(* IEC 61131-3 sources: cc_kush_rewrite/POUs, 7 files *)

(* ---- GLOBAL.st ---- *)
VAR_GLOBAL
	// Системные ФБ
	PULSE : BLINK;
	PULSE_RTRIG : R_TRIG;

	// Системные флаги
	xStateEmergencyStop : BOOL; // Система была аварийно остановлена
	xStateErrorAcceptIdle : BOOL; // Невозможно принять коэффицент шихтования по заданию оператора - сумма коэффицентов не равна 100
	xStateErrorCheckReady : BOOL; // Проверки стадии готовности к пуску провалились
	xStateAutoWorking : BOOL; // Система полностью запущена и работает в автоматическом режиме
	// Расчёт КИУМ
	ICUR_PRECENT : REAL; // Коэффициент использования установленной мощности (в процентах)
	rElectricityMeter : REAL; // Раход электроэнергии

	// Ограничение производительности
	EFFICIENCY_LIMIT_RATE : REAL := 1; // Коэффицент ограничения производительности (0-1)

	// Переменные симуляции
	SIMULATION : BOOL := TRUE;
	SIMULATION_BUNKER_WEIGHT : BOOL := FALSE; // Включение симуляции расхода и пополнения веса бункеров

	// == MODBUS РЕГИСТРЫ ДЛЯ SCADA ==
	// Массив регистров для передачи данных в SCADA систему
	awModbusInputRegisters : ARRAY [0..511] OF WORD; // Modbus Input регистры
	awModbusHoldingRegisters : ARRAY [0..511] OF WORD; // Modbus Holding регистры

	// == СИГНАЛЫ СВЯЗИ СО SCADA ==
	SCADA_HEARTBEAT : BOOL := FALSE; // Пульсирующий сигнал от SCADA (0 → 1 → 0) для контроля связи

END_VAR
VAR_GLOBAL RETAIN
	// == НАСТРОЙКИ ОСТАНОВКИ ==
	BUNKER_INSTANT_STOP : BOOL := FALSE; // Флаг мгновенной остановки бункеров (TRUE = одновременная остановка всех 3-х бункеров, FALSE = последовательная остановка)

	// == ОПЦИИ ВКЛЮЧЕНИЯ ИСТОЧНИКОВ В ГЛОБАЛЬНУЮ АВАРИЙНУЮ ОСТАНОВКУ ==
	// TRUE = источник включен в цепь глобальной аварийной остановки комплекса
	// FALSE = источник НЕ вызывает глобальную остановку

	// Датчики безопасности
	ENABLE_GLOBAL_ESTOP_ZQ : BOOL := TRUE;       // Датчики схода ленты (ZQ Alarm)
	ENABLE_GLOBAL_ESTOP_HQ : BOOL := TRUE;       // Кабель-тросовые выключатели
	ENABLE_GLOBAL_ESTOP_SQ : BOOL := FALSE;      // Концевики ограждений барабана
	ENABLE_GLOBAL_ESTOP_GS : BOOL := TRUE;      // Заштыбовка
	ENABLE_GLOBAL_ESTOP_YS : BOOL := TRUE;       // Продольный разрыв ленты
	ENABLE_GLOBAL_ESTOP_YE : BOOL := TRUE;       // Металлодетектор
	ENABLE_GLOBAL_ESTOP_QR : BOOL := FALSE;      // Датчики скорости

	// Системные сигналы
	ENABLE_GLOBAL_ESTOP_SCADA_LOSS : BOOL := FALSE;          // Потеря связи со SCADA
	ENABLE_GLOBAL_ESTOP_PROPORTION : BOOL := FALSE;          // Ошибка суммы пропорций
	ENABLE_GLOBAL_ESTOP_MOTOR_CURRENT_HH : BOOL := FALSE;    // Аварийный уровень тока (HH)
	ENABLE_GLOBAL_ESTOP_VFD_FAILURE : BOOL := TRUE;          // Авария VFD (частотного преобразователя)

	// Блокировочные зависимости (глобально)
	ENABLE_GLOBAL_ESTOP_DEPENDENCIES : BOOL := TRUE;         // Блокировочные зависимости между секциями

	// Блокировочные зависимости (индивидуально по секциям)
	// TRUE = секция останавливается при нарушении зависимостей
	// FALSE = секция НЕ останавливается при нарушении зависимостей
	ENABLE_ESTOP_DEPENDENCIES_DUMPER : BOOL := TRUE;         // Зависимости для отвалообразователя
	ENABLE_ESTOP_DEPENDENCIES_CONVEYOR : BOOL := TRUE;       // Зависимости для сборного конвейера
	ENABLE_ESTOP_DEPENDENCIES_BUNKER1 : BOOL := TRUE;        // Зависимости для бункера 1
	ENABLE_ESTOP_DEPENDENCIES_BUNKER2 : BOOL := TRUE;        // Зависимости для бункера 2
	ENABLE_ESTOP_DEPENDENCIES_BUNKER3 : BOOL := TRUE;        // Зависимости для бункера 3

	// == УСТАВКИ ==
	VFD_FREQUENCY_MAX : REAL := 50;
	VFD_FREQUENCY_STEP : REAL := 2;
	VFD_FREQUENCY_INACCURANCY : REAL := 0.5;
	VFD_FREQUENCY_SYNC_TOLERANCE : REAL := 1.5; // Допустимая разница частот для синхронизации моторов

		// == ПАРАМЕТРЫ АЦП/ЦАП ДЛЯ ЧРП ==
	VFD_ADC_MAX : INT := 27648; // Максимальный код АЦП (аналоговый вход/выход)
	VFD_ADC_MIN : INT := 0; // Минимальный код АЦП
	VFD_FREQ_MIN : REAL := 0.0; // Минимальная частота ЧРП (Гц)
	VFD_FREQ_MAX_RANGE : REAL := 50.0; // Максимальная частота для масштабирования АЦП (Гц)

	// == ПАРАМЕТРЫ ТОКА 4-20 мА ==
	VFD_CURRENT_MIN : REAL := 4.0; // Минимальный ток (мА)
	VFD_CURRENT_MAX : REAL := 20.0; // Максимальный ток (мА)
	VFD_CURRENT_ALARM_LL : REAL := 3.8; // Аварийно низкий уровень тока (обрыв линии)
	VFD_CURRENT_ALARM_L : REAL := 4.5; // Низкий уровень тока
	VFD_CURRENT_ALARM_H : REAL := 19.5; // Высокий уровень тока
	VFD_CURRENT_ALARM_HH : REAL := 20.2; // Аварийно высокий уровень тока (перегрузка)

	// == ПАРАМЕТРЫ ДИАПАЗОНА ТЕМПЕРАТУР ==
	TEMP_BEARING_MIN : REAL := 0.0; // Минимальная температура подшипникового узла (°C)
	TEMP_BEARING_MAX : REAL := 100.0; // Максимальная температура подшипникового узла (°C)

	// Настройка виброобрушения
	VIBRATOR_SETTINGS : ST_BunkerVibratorSettings := (
		TIME_ACTIVE := T#15S,
		TIME_PAUSE_VIBRATOR := T#30S,
		TIME_PAUSE_FB := T#30S,
		COUNT_CYCLE := 3
		);

	// Время шага последовательного запуска вибраторов (задержка между запуском каждого следующего вибратора в фазе ACTIVE)
	TIME_VIBRATOR_SEQUENTIAL_START_STEP : TIME := T#4S;

	// Настройка пневмообрушения
	PNEUMO_SETTINGS : ST_BunkerVibratorSettings := (
		TIME_ACTIVE := T#10S,
		TIME_PAUSE_VIBRATOR := T#10S,
		TIME_PAUSE_FB := T#30S,
		COUNT_CYCLE := 3
		);

	// Опция плавного задания частоты
	VFD_SMOOTH_SET_FREQUENCY : BOOL := FALSE;

	// Таймеры последовательного запуска механизмов в автоматическом режиме
	TIME_AFTER_START_DUMPER : TIME := T#120S; // Время ожидания после запуска отвалообразователя
	TIME_AFTER_START_CONVEYOR : TIME := T#120S; // Время ожидания после запуска конвейера
	TIME_AFTER_START_BUNKER_1 : TIME := T#120S; // Время ожидания после запуска бункера 1
	TIME_AFTER_START_BUNKER_2 : TIME := T#120S; // Время ожидания после запуска бункера 2
	TIME_AFTER_START_BUNKER_3 : TIME := T#120S; // Время ожидания после запуска бункера 3

	// Таймеры контроля выполнения команд (тайм-ауты)
	TIME_TIMEOUT_START_DUMPER_CONVEYOR : TIME := T#30S; // Тайм-аут запуска моторов конвейера отвалообразователя (STARTING → WORK)
	TIME_TIMEOUT_START_DUMPER_ROTATION : TIME := T#20S; // Тайм-аут запуска моторов поворота отвалообразователя (STARTING → WORK)
	TIME_TIMEOUT_START_CONVEYOR : TIME := T#30S; // Тайм-аут запуска моторов сборного конвейера (STARTING → WORK)
	TIME_TIMEOUT_START_BUNKER : TIME := T#20S; // Тайм-аут запуска вибропитателей бункера (STARTING → WORK)
	TIME_TIMEOUT_STOP_DUMPER_CONVEYOR : TIME := T#30S; // Тайм-аут остановки моторов конвейера отвалообразователя (STOPPING → IDLE)
	TIME_TIMEOUT_STOP_DUMPER_ROTATION : TIME := T#20S; // Тайм-аут остановки моторов поворота отвалообразователя (STOPPING → IDLE)
	TIME_TIMEOUT_STOP_CONVEYOR : TIME := T#30S; // Тайм-аут остановки моторов сборного конвейера (STOPPING → IDLE)
	TIME_TIMEOUT_STOP_BUNKER : TIME := T#20S; // Тайм-аут остановки вибропитателей бункера (WORK → IDLE)

	// Таймер ожидания восстановления потерянной обратной связи VFD во время работы
	TIME_TIMEOUT_VFD_FEEDBACK_LOST : TIME := T#3S; // Если обратная связь VFD пропала во время WORK и не вернулась в течение этого времени → аварийная остановка

	// Таймер ожидания пропавшего сигнала обратной связи работы механизма
	TIME_WAITING_FEEDBACK : TIME := T#0S;

	// == ПАРАМЕТРЫ СВЯЗИ СО SCADA ==
	SCADA_HEARTBEAT_TIMEOUT : TIME := T#5S; // Таймаут отсутствия изменений heartbeat сигнала (потеря связи)

	// Таймаут контроля суммы пропорций в режиме WORK
	BUNKER_PROPORTION_SUM_TIMEOUT : TIME := T#20S; // Время ожидания корректировки суммы пропорций оператором (сумма должна быть = 100%)

	// Скорость конвейера
	CONVEYOR_DEAFULT_SPEED : REAL := -1;

	// Температура подшипникового узла мотора вибропитателя
	MOTOR_VIBFEEDER_TEMP_POINTS : ST_AlarmSetpoints := (
		LL_Value := -1,
		L_Value := -1,
		H_Value := -1,
		HH_Value := -1);
	// Ток мотора вибропитателя
	MOTOR_VIBFEEDER_CURRENT_POINTS : ST_AlarmSetpoints := (
		LL_Value := -1,
		L_Value := -1,
		H_Value := -1,
		HH_Value := -1);
	// Ток мотора вибратора
	MOTOR_VIBRATOR_CURRENT_POINTS : ST_AlarmSetpoints := (
		LL_Value := -1,
		L_Value := -1,
		H_Value := -1,
		HH_Value := -1);
	// Ток мотора конвейера отвалообразователя
	MOTOR_CONVEYOR_CURRENT_POINTS : ST_AlarmSetpoints := (
		LL_Value := -1,
		L_Value := -1,
		H_Value := -1,
		HH_Value := -1);
	// Ток мотора конвейера сборного
	MOTOR_CONVEYOR_PREFABRICATED_CURRENT_POINTS : ST_AlarmSetpoints := (
		LL_Value := -1,
		L_Value := -1,
		H_Value := -1,
		HH_Value := -1);
	// Ток мотора поворота отвалообразователя
	MOTOR_ROTATION_CURRENT_POINTS : ST_AlarmSetpoints := (
		LL_Value := -1,
		L_Value := -1,
		H_Value := -1,
		HH_Value := -1);

	// Предпусковая сигнализация конвейера отвалообразователя
	DUMPER_CONVEYOR_PRESTART_ALARM_SETTINGS : ST_PreStartAlarmSettings := (
		OPTION_ENABLE := TRUE, // Опция на включение ППЗ в алгоритм
		TIME_FIRST_SIGNAL := T#3S, // Время звучания первого сигнала
		TIME_FIRST_SIGNAL_PAUSE := T#3S, // Пауза после первого сигнала
		TIME_SECOND_SIGNAL := T#3S, // Время звучания второго сигнала
		TIME_SECOND_SIGNAL_PAUSE := T#3S); // Пауза после втотрого сигнала

	// Предпусковая сигнализация сборного конвейера
	CONVEYOR_PRESTART_ALARM_SETTINGS : ST_PreStartAlarmSettings := (
		OPTION_ENABLE := TRUE, // Опция на включение ППЗ в алгоритм
		TIME_FIRST_SIGNAL := T#3S, // Время звучания первого сигнала
		TIME_FIRST_SIGNAL_PAUSE := T#3S, // Пауза после первого сигнала
		TIME_SECOND_SIGNAL := T#3S, // Время звучания второго сигнала
		TIME_SECOND_SIGNAL_PAUSE := T#3S); // Пауза после втотрого сигнала

	// Световая индикация Гц
	ANNUNCIATOR_LIGHT_HZ : REAL := 2;

	// Частота мотора конвейера
	MOTOR_FREQUENCY_CONVEYOR : REAL := 50;
	// Частота мотора конвейера отвалообразователя
	MOTOR_FREQUENCY_DUMPER_CONVEYOR : REAL := 50;
	// Частота мотора поворота отвалообразователя
	MOTOR_FREQUENCY_DUMPER_ROTATION : REAL := -1;

	BUNKER_MINIMAL_WEIGHT :REAL := 0; // Уставка минимального веса бункера. Результат <= считывается алгоритмом как пустой бункер.

	// Уставки бункера
	PNEUMATIC_COLLAPSE_TIME : TIME := T#0S; // Уставка времени таймера пневмообрушения
	BUNKER_WORK_PRECENT_1 : REAL; // Уставка пропорции шихтования для бункера 1
	BUNKER_WORK_PRECENT_2 : REAL; // Уставка пропорции шихтования для бункера 2
	BUNKER_WORK_PRECENT_3 : REAL; // Уставка пропорции шихтования для бункера 3
	BUNKER_VIBFEEDER_START_FREQUENCY : REAL := 10.0; // Минимальная частота для запуска вибропитателей (Гц)
	BUNKER_VIBFEEDER_FREQUENCY_TARGET_SUM : REAL := 50.0; // Целевая суммарная частота вибропитателей (Гц)
    BUNKER_ENABLE_PID : BOOL := FALSE;
    BUNKER_ENABLE_PROPORTION_MONITORING : BOOL := FALSE;

	// == КОНТРОЛЬ МИНИМАЛЬНОЙ И МАКСИМАЛЬНОЙ ЧАСТОТЫ ВИБРОПИТАТЕЛЯ (ДЛЯ ПИД-РЕГУЛЯТОРА) ==
	BUNKER_VIBFEEDER_MIN_FREQUENCY_LIMIT : REAL := 5.0; // Минимальная допустимая частота вибропитателя (Гц) - при достижении этой уставки запускается таймер аварии
	BUNKER_VIBFEEDER_MIN_FREQUENCY_TIMEOUT : TIME := T#30S; // Время задержки перед аварийной остановкой при достижении минимальной частоты
	BUNKER_VIBFEEDER_MAX_FREQUENCY_LIMIT : REAL := 50.0; // Максимальная допустимая частота вибропитателя (Гц) - при достижении этой уставки запускается таймер аварии
	BUNKER_VIBFEEDER_MAX_FREQUENCY_TIMEOUT : TIME := T#30S; // Время задержки перед аварийной остановкой при достижении максимальной частоты

	// Ручное задание частоты на бункер (работает в ручном режиме управления)
	BUNKER_1_FREQ_VIBFEEDER : REAL := 30;
	BUNKER_1_FREQ_VIBRATOR : REAL := 30;
	BUNKER_2_FREQ_VIBFEEDER : REAL := 30;
	BUNKER_2_FREQ_VIBRATOR : REAL := 30;
	BUNKER_3_FREQ_VIBFEEDER : REAL := 30;
	BUNKER_3_FREQ_VIBRATOR : REAL := 30;

	// Светофор бункера
	BUNKER_WEIGHT_LIGHT_RED : REAL := 90; // Уставка веса бункера для красного светофора
	BUNKER_WEIGHT_LIGHT_YELLOW : REAL := 80; // Уставка веса бункера для жёлтого светофора
	BUNKER_WEIGHT_LIGHT_GREEN : REAL := 50; // Уставка веса бункера для зелёного светофора

	BUNKER_WEIGHT_LIGHT_RED_SPECIAL : REAL := 10; // Уставка веса бункера для красного светофора, когда сырье закончилось и требуется остановить подачу материала в остальные бункеры для будущего алгоритма опустошения

	// Константы
	AMOUNT_BUNKER_MOTOR_VIBFEEDER : INT := 2;
	AMOUNT_BUNKER_MOTOR_VIBRATOR : INT := 4;

	// == УСТАВКИ ЗАДЕРЖКИ СРАБАТЫВАНИЯ ДАТЧИКОВ БЕЗОПАСНОСТИ ==
	// Таймеры задержки для датчиков отвалообразователя (Dumper)
	TIME_DELAY_SENSOR_DUMPER_ZQ_ALARM : TIME := T#3S;   // Задержка срабатывания датчика схода ленты (Alarm)
	TIME_DELAY_SENSOR_DUMPER_ZQ_WARNING : TIME := T#0S; // Задержка срабатывания датчика схода ленты (Warning)
	TIME_DELAY_SENSOR_DUMPER_HQ : TIME := T#0S;         // Задержка срабатывания кабель-тросового выключателя
	TIME_DELAY_SENSOR_DUMPER_SQ : TIME := T#0S;         // Задержка срабатывания датчика ограждения барабана
	TIME_DELAY_SENSOR_DUMPER_GS : TIME := T#3S;         // Задержка срабатывания датчика заштыбовки
	TIME_DELAY_SENSOR_DUMPER_YS : TIME := T#3S;         // Задержка срабатывания датчика продольного разрыва
	TIME_DELAY_SENSOR_DUMPER_QR : TIME := T#0S;         // Задержка срабатывания датчика скорости

	// Таймеры задержки для датчиков сборного конвейера (Conveyor)
	TIME_DELAY_SENSOR_CONVEYOR_ZQ_ALARM : TIME := T#3S;   // Задержка срабатывания датчика схода ленты (Alarm)
	TIME_DELAY_SENSOR_CONVEYOR_ZQ_WARNING : TIME := T#0S; // Задержка срабатывания датчика схода ленты (Warning)
	TIME_DELAY_SENSOR_CONVEYOR_HQ : TIME := T#0S;         // Задержка срабатывания кабель-тросового выключателя
	TIME_DELAY_SENSOR_CONVEYOR_SQ : TIME := T#0S;         // Задержка срабатывания датчика ограждения барабана
	TIME_DELAY_SENSOR_CONVEYOR_GS : TIME := T#3S;         // Задержка срабатывания датчика заштыбовки
	TIME_DELAY_SENSOR_CONVEYOR_YS : TIME := T#3S;         // Задержка срабатывания датчика продольного разрыва
	TIME_DELAY_SENSOR_CONVEYOR_YE : TIME := T#0S;         // Задержка срабатывания металлодетектора
	TIME_DELAY_SENSOR_CONVEYOR_QR : TIME := T#0S;         // Задержка срабатывания датчика скорости
END_VAR

(* ---- FB_ConveyorWeight.st ---- *)
FUNCTION_BLOCK FB_ConveyorWeight
VAR_INPUT
	wModbusReg : ARRAY [0..22] OF WORD;
END_VAR
VAR_OUTPUT
	qrWeight : REAL; 			//	0x0 Производительность
	qrSpeed : REAL; 			//	0x2 Скорость
	qrWorkLoad : REAL; 			//	0x4 Погонная нагрузка
	qrVoltageTenso_1 : REAL; 	//	0x6 Текущее напряжение тензодатчика 1
	qrVoltageTenso_2 : REAL; 	//	0x8 Текущее напряжение тензодатчика 2
	qrVoltageTenso_3 : REAL; 	//	0xA Текущее напряжение тензодатчика 3
	qrVoltageTenso_4 : REAL; 	//	0xC Текущее напряжение тензодатчика 4
 	qrCounterShift : REAL;		//	0xE Счётчик: смена
	qrCounterDay : REAL;		//	0xE Счётчик: смена
	qrCounterMonth : REAL;		//	0xE Счётчик: смена
	qrCounterCommon : REAL;		//	0xE Счётчик: смена

END_VAR
VAR
END_VAR

END_FUNCTION_BLOCK

(* ---- FB_DumperControl.st ---- *)
FUNCTION_BLOCK FB_DumperControl
VAR_INPUT
	Dumper : REFERENCE TO ST_Dumper;
	xLocalMode : BOOL; // TRUE = местный режим (ПМУ), FALSE = дистанционный режим (SCADA)
	xStart : BOOL; // Команда запуска отвалообразователя (дистанционный режим)
	xStop : BOOL; // Команда остановки (дистанционный режим)
	xEmergencyStop : BOOL; // Аварийная остановка
	xReset : BOOL; // Сброс в начальное состояние
	xDisableAutoEmergencyStop : BOOL; // Отключение автоматических аварийных остановок по датчикам безопасности
END_VAR
VAR_OUTPUT
	eStage : E_StageWithPreStartAlarm; // Текущая стадия
	eStageToSCADA : E_ScadaStatesDevice; // Передача состояния скаде
END_VAR
VAR
	// Состояния
	STAGE : E_StageWithPreStartAlarm := E_StageWithPreStartAlarm.IDLE;

	// Объединенные команды (ПМУ или SCADA в зависимости от режима)
	xStartCommand : BOOL; // Фактическая команда запуска (из ПМУ или SCADA)
	xStopCommand : BOOL; // Фактическая команда остановки (из ПМУ или SCADA)

	// Целевые частоты для моторов
	rTargetFreqConv1 : REAL := 0.0;
	rTargetFreqConv2 : REAL := 0.0;
	rTargetFreqRot1 : REAL := 0.0;
	rTargetFreqRot2 : REAL := 0.0;

	// Переменные синхронизации моторов конвейера
	xVFDsReady : BOOL; // Оба ЧРП конвейера готовы и запущены
	xFrequenciesSynchronized : BOOL; // Частоты синхронизированы в пределах допуска
	xConditionToProceed : BOOL; // Общее условие для продолжения разгона

	// Подстадии запуска (для последовательного включения тормозов и VFD)
	nStartingSubstage : INT := 0;
	// 0 - RELEASE_BRAKE: Отпускание тормозов
	// 1 - WAIT_BRAKE_FEEDBACK: Ожидание обратной связи тормозов
	// 2 - START_VFD: Запуск VFD
	// 3 - RAMPING: Разгон частоты до рабочей

	// Подстадии остановки (для последовательного выключения VFD и тормозов)
	nStoppingSubstage : INT := 0;
	// 0 - Нормальная работа
	// 1 - SET_FREQUENCY_ZERO: Установка частоты 0 на аналоговый выход
	// 2 - WAIT_FREQUENCY_ZERO: Ожидание подтверждения частоты 0 с аналогового входа
	// 3 - STOP_VFD: Остановка VFD (снятие команды пуска)
	// 4 - WAIT_VFD_STOP: Ожидание остановки VFD (обратная связь)
	// 5 - ACTIVATE_BRAKE: Активация тормозов
	// 6 - WAIT_BRAKE_FEEDBACK: Ожидание обратной связи тормозов

	// Состояние схемы контакторов (TRUE = схема собрана, FALSE = схема разобрана)
	xCircuitBuilt : BOOL := FALSE;
	xCircuitBuiltRotation : BOOL := FALSE;

	// Таймеры контроля выполнения команд
	fbTimerStarting : TON; // Тайм-аут запуска (STARTING → WORK)
	fbTimerStopping : TON; // Тайм-аут остановки (WORK → IDLE)
	fbTimerRotation : TON; // Тайм-аут выполнения команд поворота
	// Таймер на работу тормоза
	tonTimerEnableBreakerConveyor : TON; // Задержка включения тормоза на конвейере
	tonTimerEnableBreakerRotation : TON; // Задержка включения тормоза на повороте

	// == Управление поворотом ==
	xRotationLeftActive : BOOL; // Поворот влево активен
	xRotationRightActive : BOOL; // Поворот вправо активен
	nRotationSubstage : INT := 0; // Подстадии поворота
	// 0 - IDLE: Нет активного поворота
	// 1 - RELEASE_BRAKE: Отпускание тормоза поворота
	// 2 - WAIT_BRAKE_FEEDBACK: Ожидание обратной связи тормоза
	// 3 - START_VFD: Запуск VFD поворота
	// 4 - WORKING: Моторы поворота работают
	// 5 - SET_FREQUENCY_ZERO: Установка частоты 0 на аналоговый выход
	// 6 - WAIT_FREQUENCY_ZERO: Ожидание подтверждения частоты 0 с аналогового входа
	// 7 - STOP_VFD: Остановка VFD поворота (снятие команды пуска)
	// 8 - WAIT_VFD_STOP: Ожидание остановки VFD (обратная связь)
	// 9 - ACTIVATE_BRAKE: Активация тормоза

	simInit : BOOL;
	i : INT;
END_VAR

// ========================================
// FB_DumperControl - Управление отвалообразователем
// ========================================
//
// РЕЖИМЫ УПРАВЛЕНИЯ:
//
// 1. МЕСТНЫЙ РЕЖИМ (xLocalMode = TRUE):
//    - Команды берутся с кнопок ПМУ (Dumper.fbBtnStart, fbBtnStop)
//    - Конвейер: ПУСК/СТОП по фронтам кнопок
//    - Поворот: работает пока кнопка ЗАЖАТА (fbBtnTurnLeft/Right)
//    - Автоматически устанавливает eStateRemote = Manual
//
// 2. ДИСТАНЦИОННЫЙ РЕЖИМ (xLocalMode = FALSE):
//    - Команды берутся из входов ФБ (xStart, xStop)
//    - Конвейер: ПУСК/СТОП по входам ФБ
//    - Поворот: импульсные команды через Dumper.cmdTurnLeft/Right/Stop
//    - Режим устанавливается через SCADA (Manual/Remote/Auto)
//
// УПРАВЛЕНИЕ КОНВЕЙЕРОМ:
// - ПУСК: включение конвейеров отвалообразователя
// - СТОП: плавная остановка с последовательным выключением VFD и тормозов
//
// УПРАВЛЕНИЕ ПОВОРОТОМ:
// - Местный: поворот пока кнопка зажата (отпустили - остановка)
// - Дистанционный: импульсные команды от SCADA
// - Блокировка по концевикам (fbEndSwitchLeft/Right):
//   * Если концевик сработал (qxSignal = FALSE), команда поворота в эту сторону игнорируется
//   * Поворот автоматически останавливается при достижении концевика
//
// ========================================

// ========================================
// ИНИЦИАЛИЗАЦИЯ СИГНАЛОВ
// ========================================

// ПМУ - СТАРТ
Dumper.fbBtnStart(
	ixSignal := , // Подключить физический вход
	xEnableRattlingFilter := TRUE,
	tStabilityTime := T#100MS
);

// ПМУ - СТОП
Dumper.fbBtnStop(
	ixSignal := , // Подключить физический вход
	xEnableRattlingFilter := TRUE,
	tStabilityTime := T#100MS
);

// ПМУ - Аварийная остановка
Dumper.fbBtnEmergencyStop(
	ixSignal := , // Подключить физический вход
	xEnableRattlingFilter := TRUE,
	tStabilityTime := T#100MS
);

// ПМУ Поворот влево/вправо
Dumper.fbBtnTurnLeft(
	ixSignal := , // Подключить физический вход
	xEnableRattlingFilter := TRUE,
	tStabilityTime := T#100MS
);

Dumper.fbBtnTurnRight(
	ixSignal := , // Подключить физический вход
	xEnableRattlingFilter := TRUE,
	tStabilityTime := T#100MS
);

Dumper.fbEndSwitchLeft(
	ixSignal := , // Подключить физический вход
	xEnableRattlingFilter := TRUE,
	tStabilityTime := T#100MS
);

Dumper.fbEndSwitchRight(
	ixSignal := , // Подключить физический вход
	xEnableRattlingFilter := TRUE,
	tStabilityTime := T#100MS
);

// Сигналы тормозоов (Обратная связь)
Dumper.fbBreakerConveyor(
	ixSignal := , // Физ. сигнал
	xEnableRattlingFilter := TRUE);

Dumper.fbBreakerRotation(
	ixSignal := , // Физ. сигнал
	xEnableRattlingFilter := TRUE);

// Двигатели конвейера
FOR i := 1 TO 2 BY 1 DO
	Dumper.MotorConveyor[i].fbStateKM(
		ixSignal := , // Состояние контактора
		xEnableRattlingFilter := TRUE
	);

	Dumper.MotorConveyor[i].fbStatorOverheat(
		ixSignal := , // Перегрев статора
		xEnableRattlingFilter := TRUE
	);

	Dumper.MotorConveyor[i].fbStateQF(
		ixSignal := , // Автомат. выключатель
		xEnableRattlingFilter := TRUE
	);

	Dumper.MotorConveyor[i].VFD.fbStateFailure(
		ixSignal := , // ЧРП - ошибка
		xEnableRattlingFilter := TRUE
	);

	Dumper.MotorConveyor[i].VFD.fbStateRdyToStart(
		ixSignal := , // ЧРП - Готовность
		xEnableRattlingFilter := TRUE
	);

	Dumper.MotorConveyor[i].VFD.fbStateIsWorking(
		ixSignal := , // ЧРП - Работа
		xEnableRattlingFilter := TRUE
	);

	// Инициализация устройств
	Dumper.MotorConveyor[i].Device(
		ixFeedback := Dumper.MotorConveyor[i].fbStateKM.qxSignal,
		xEnableFeedback := TRUE
	);

	// ЧРП
	Dumper.MotorConveyor[i].VFD.Device(
		ixFeedback := Dumper.MotorConveyor[i].VFD.fbStateIsWorking.qxSignal,
		xEnableFeedback := TRUE
	);

	// VFD.qxStart теперь управляется напрямую в алгоритме (TRUE = ПУСК, FALSE = СТОП)

	// Диагностика тока
	Dumper.MotorConveyor[i].VFD.fbRangeDiagnostic(
		irValue := Dumper.MotorConveyor[i].VFD.wMotorCurrent.rTag,
		irSetpointL := MOTOR_CONVEYOR_CURRENT_POINTS.L_Value,
		irSetpointLL := MOTOR_CONVEYOR_CURRENT_POINTS.LL_Value,
		irSetpointH := MOTOR_CONVEYOR_CURRENT_POINTS.H_Value,
		irSetpointHH := MOTOR_CONVEYOR_CURRENT_POINTS.HH_Value,
		ixEnable := TRUE
	);

	// Аналоговый вход ЧРП (чтение текущей частоты)
	Dumper.MotorConveyor[i].VFD.fbAnalogInput(
		xSimulation := SIMULATION,
		iADC_Code := Dumper.MotorConveyor[i].VFD.nActualFrequencyADC,
		refEngValue := Dumper.MotorConveyor[i].VFD.rActualFrequency,
		refSimValue := Dumper.MotorConveyor[i].VFD.rSimulatedFrequency,
		rAlarm_LL := VFD_CURRENT_ALARM_LL,
		rAlarm_L := VFD_CURRENT_ALARM_L,
		rAlarm_H := VFD_CURRENT_ALARM_H,
		rAlarm_HH := VFD_CURRENT_ALARM_HH,
		iADC_Max := VFD_ADC_MAX,
		iADC_Min := VFD_ADC_MIN,
		rEngValue_Max := VFD_FREQ_MAX_RANGE,
		rEngValue_Min := VFD_FREQ_MIN,
		rCurrent_Max := VFD_CURRENT_MAX,
		rCurrent_Min := VFD_CURRENT_MIN
	);

	// Аналоговый выход ЧРП (задание частоты)
	Dumper.MotorConveyor[i].VFD.fbAnalogOutput(
		xEnable := Dumper.MotorConveyor[i].VFD.Device.qxActive,
		rEngValue := Dumper.MotorConveyor[i].VFD.Frequency.qrCurrentFrequency,
		rEngValue_Max := VFD_FREQ_MAX_RANGE,
		rEngValue_Min := VFD_FREQ_MIN,
		rCurrent_Max := VFD_CURRENT_MAX,
		rCurrent_Min := VFD_CURRENT_MIN,
		iDAC_Max := VFD_ADC_MAX,
		iDAC_Min := VFD_ADC_MIN,
		rAlarm_LL := VFD_CURRENT_ALARM_LL,
		rAlarm_L := VFD_CURRENT_ALARM_L,
		rAlarm_H := VFD_CURRENT_ALARM_H,
		rAlarm_HH := VFD_CURRENT_ALARM_HH,
		xEnableClamp := TRUE
	);
	Dumper.MotorConveyor[i].VFD.nSetOutSignalToModule := Dumper.MotorConveyor[i].VFD.fbAnalogOutput.iDAC_Code;
END_FOR;

// Двигатели поворота
FOR i := 1 TO 2 BY 1 DO
	Dumper.MotorRotation[i].fbStateKM(
		ixSignal := , // Состояние контактора
		xEnableRattlingFilter := TRUE
	);

	Dumper.MotorRotation[i].fbStatorOverheat(
		ixSignal := , // Перегрев статора
		xEnableRattlingFilter := TRUE
	);

	Dumper.MotorRotation[i].fbStateQF(
		ixSignal := , // Автомат. выключатель
		xEnableRattlingFilter := TRUE
	);

	Dumper.MotorRotation[i].VFD.fbStateFailure(
		ixSignal := , // ЧРП - ошибка
		xEnableRattlingFilter := TRUE
	);

	Dumper.MotorRotation[i].VFD.fbStateRdyToStart(
		ixSignal := , // ЧРП - Готовность
		xEnableRattlingFilter := TRUE
	);

	Dumper.MotorRotation[i].VFD.fbStateIsWorking(
		ixSignal := , // ЧРП - Работа
		xEnableRattlingFilter := TRUE
	);

	Dumper.MotorRotation[i].fbRotationStatus(
		ixSignal := , // Статус вращения
		xEnableRattlingFilter := TRUE
	);

	// Инициализация устройств
	Dumper.MotorRotation[i].Device(
		ixFeedback := Dumper.MotorRotation[i].fbStateKM.qxSignal,
		xEnableFeedback := TRUE
	);

	// ЧРП
	Dumper.MotorRotation[i].VFD.Device(
		ixFeedback := Dumper.MotorRotation[i].VFD.fbStateIsWorking.qxSignal,
		xEnableFeedback := TRUE
	);

	// VFD.qxStart теперь управляется напрямую в алгоритме (TRUE = ПУСК, FALSE = СТОП)

	// Диагностика тока
	Dumper.MotorRotation[i].VFD.fbRangeDiagnostic(
		irValue := Dumper.MotorRotation[i].VFD.wMotorCurrent.rTag,
		irSetpointL := MOTOR_ROTATION_CURRENT_POINTS.L_Value,
		irSetpointLL := MOTOR_ROTATION_CURRENT_POINTS.LL_Value,
		irSetpointH := MOTOR_ROTATION_CURRENT_POINTS.H_Value,
		irSetpointHH := MOTOR_ROTATION_CURRENT_POINTS.HH_Value,
		ixEnable := TRUE
	);

	// Аналоговый вход ЧРП (чтение текущей частоты)
	Dumper.MotorRotation[i].VFD.fbAnalogInput(
		xSimulation := SIMULATION,
		iADC_Code := Dumper.MotorRotation[i].VFD.nActualFrequencyADC,
		refEngValue := Dumper.MotorRotation[i].VFD.rActualFrequency,
		refSimValue := Dumper.MotorRotation[i].VFD.rSimulatedFrequency,
		rAlarm_LL := VFD_CURRENT_ALARM_LL,
		rAlarm_L := VFD_CURRENT_ALARM_L,
		rAlarm_H := VFD_CURRENT_ALARM_H,
		rAlarm_HH := VFD_CURRENT_ALARM_HH,
		iADC_Max := VFD_ADC_MAX,
		iADC_Min := VFD_ADC_MIN,
		rEngValue_Max := VFD_FREQ_MAX_RANGE,
		rEngValue_Min := VFD_FREQ_MIN,
		rCurrent_Max := VFD_CURRENT_MAX,
		rCurrent_Min := VFD_CURRENT_MIN
	);

	// Аналоговый выход ЧРП (задание частоты)
	Dumper.MotorRotation[i].VFD.fbAnalogOutput(
		xEnable := Dumper.MotorRotation[i].VFD.Device.qxActive,
		rEngValue := Dumper.MotorRotation[i].VFD.Frequency.qrCurrentFrequency,
		rEngValue_Max := VFD_FREQ_MAX_RANGE,
		rEngValue_Min := VFD_FREQ_MIN,
		rCurrent_Max := VFD_CURRENT_MAX,
		rCurrent_Min := VFD_CURRENT_MIN,
		iDAC_Max := VFD_ADC_MAX,
		iDAC_Min := VFD_ADC_MIN,
		rAlarm_LL := VFD_CURRENT_ALARM_LL,
		rAlarm_L := VFD_CURRENT_ALARM_L,
		rAlarm_H := VFD_CURRENT_ALARM_H,
		rAlarm_HH := VFD_CURRENT_ALARM_HH,
		xEnableClamp := TRUE
	);
	Dumper.MotorRotation[i].VFD.nSetOutSignalToModule := Dumper.MotorRotation[i].VFD.fbAnalogOutput.iDAC_Code;
END_FOR;

// Датчики безопасности
FOR i := 1 TO 4 BY 1 DO
	Dumper.fbZQAlarm[i](
		ixSignal := ,
		xEnableRattlingFilter := TRUE
	);

	Dumper.fbZQWarning[i](
		ixSignal := ,
		xEnableRattlingFilter := TRUE
	);

	Dumper.fbHQ_IsOk[i](
		ixSignal := ,
		xEnableRattlingFilter := TRUE
	);
END_FOR;

FOR i := 1 TO 2 BY 1 DO
	Dumper.fbSQ_IsOk[i](
		ixSignal := ,
		xEnableRattlingFilter := TRUE
	);

	Dumper.fbQR[i](
		ixSignal := ,
		xEnableRattlingFilter := FALSE // Только edge detection
	);
END_FOR;

Dumper.fbGS1(
	ixSignal := ,
	xEnableRattlingFilter := TRUE
);

Dumper.fbYS1(
	ixSignal := ,
	xEnableRattlingFilter := TRUE
);

// ========================================
// ПРЕДПУСКОВАЯ СИГНАЛИЗАЦИЯ
// ========================================

Dumper.fbPreStartAlarm(
	ixStart := STAGE = PRESTART_ALARM,
	ixStop := xStopCommand OR xReset,
	itFirstSignal := DUMPER_CONVEYOR_PRESTART_ALARM_SETTINGS.TIME_FIRST_SIGNAL,
	itPauseAfterFirst := DUMPER_CONVEYOR_PRESTART_ALARM_SETTINGS.TIME_FIRST_SIGNAL_PAUSE,
	itSecondSignal := DUMPER_CONVEYOR_PRESTART_ALARM_SETTINGS.TIME_SECOND_SIGNAL,
	itPauseAfterSecond := DUMPER_CONVEYOR_PRESTART_ALARM_SETTINGS.TIME_SECOND_SIGNAL_PAUSE,
	qxAlarmPower => Dumper.xHLA
);

// Световая сигнализация во время активной работы поворота
// xHLA включается как при предпусковой сигнализации, так и при повороте
Dumper.xHLA := Dumper.fbPreStartAlarm.qxAlarmPower OR (nRotationSubstage = 4);

Dumper.xStateEnable := STAGE = E_StageWithPreStartAlarm.WORK;
Dumper.xStateStarting := STAGE = E_StageWithPreStartAlarm.STARTING OR STAGE = PRESTART_ALARM;

// ========================================
// ОПРЕДЕЛЕНИЕ СОСТОЯНИЙ ДЛЯ SCADA
// ========================================

// Проверка ошибок оборудования
IF FC_Dumper_GetErrorCommon(Dumper := Dumper) THEN
	Dumper.xStateFailure := TRUE;
END_IF;

// Проверка предупреждений:
// 1. Датчики схода ленты ZQ - уровень Warning
// 2. Контроль тока моторов - уровень L или H
Dumper.xStateWarning := NOT Dumper.fbZQWarning[1].qxSignal
                     OR NOT Dumper.fbZQWarning[2].qxSignal
                     OR NOT Dumper.fbZQWarning[3].qxSignal
                     OR NOT Dumper.fbZQWarning[4].qxSignal
                     OR Dumper.MotorConveyor[1].VFD.fbRangeDiagnostic.qxWarningActive
                     OR Dumper.MotorConveyor[2].VFD.fbRangeDiagnostic.qxWarningActive
                     OR Dumper.MotorRotation[1].VFD.fbRangeDiagnostic.qxWarningActive
                     OR Dumper.MotorRotation[2].VFD.fbRangeDiagnostic.qxWarningActive;

// ========================================
// ОБРАБОТКА ОСТАНОВКИ И СБРОСА
// ========================================

// Сброс в начальное состояние
IF xReset THEN
	Dumper.xStateFailure := FALSE;
END_IF

// Штатная остановка - запускается при получении команды xStop
// Обрабатывается через подстадии в режиме WORK

// ========================================
// ВЫБОР ИСТОЧНИКА КОМАНД (ПМУ ИЛИ SCADA)
// ========================================

// В местном режиме (xLocalMode = TRUE) - команды берутся с ПМУ (кнопки)
// В дистанционном режиме (xLocalMode = FALSE) - команды берутся из SCADA (входы ФБ)
IF xLocalMode THEN
	// Местный режим - команды с ПМУ
	xStartCommand := Dumper.fbBtnStart.qxRisingEdge; // ПУСК по фронту кнопки
	xStopCommand := Dumper.fbBtnStop.qxRisingEdge;   // СТОП по фронту кнопки
ELSE
	// Дистанционный режим - команды из SCADA
	xStartCommand := xStart;
	xStopCommand := xStop;
END_IF;

// ========================================
// АВТОМАТ ПУСКА ОТВАЛООБРАЗОВАТЕЛЯ
// ========================================

// ПРИОРИТЕТНАЯ ПРОВЕРКА АВАРИЙНОЙ ОСТАНОВКИ
// Аварийная остановка имеет наивысший приоритет и срабатывает в любой стадии
// 1. Внешний сигнал аварийной остановки (от SCADA или системы)
// 2. Кнопка аварийной остановки на ПМУ (NC контакт: FALSE = кнопка нажата)
IF xEmergencyStop OR NOT Dumper.fbBtnEmergencyStop.qxSignal THEN
	STAGE := E_StageWithPreStartAlarm.ERROR;
END_IF;

// КРИТИЧЕСКИЕ ОШИБКИ ДАТЧИКОВ БЕЗОПАСНОСТИ
// При срабатывании датчиков безопасности немедленная аварийная остановка,
// если секция НЕ в IDLE (т.е. находится в процессе работы или запуска)
// Блокируется через вход xDisableAutoEmergencyStop
IF FC_Dumper_GetErrorSensors(Dumper := Dumper)
   AND STAGE <> E_StageWithPreStartAlarm.IDLE
   AND NOT xDisableAutoEmergencyStop
THEN
	STAGE := E_StageWithPreStartAlarm.ERROR;
END_IF;

// ПРОВЕРКА ТАЙМ-АУТОВ ВЫПОЛНЕНИЯ КОМАНД
// Тайм-аут запуска: не удалось запустить секцию за установленное время
IF fbTimerStarting.Q THEN
	STAGE := E_StageWithPreStartAlarm.ERROR;
END_IF;

// Тайм-аут остановки: не удалось остановить секцию за установленное время
IF fbTimerStopping.Q THEN
	STAGE := E_StageWithPreStartAlarm.ERROR;
END_IF;

// Тайм-аут поворота: не удалось выполнить команду поворота за установленное время
IF fbTimerRotation.Q THEN
	STAGE := E_StageWithPreStartAlarm.ERROR;
	nRotationSubstage := 0; // Сброс подстадии поворота
END_IF;

CASE STAGE OF
	E_StageWithPreStartAlarm.IDLE:
		// Сброс целевой частоты
		rTargetFreqConv1 := 0.0;
		rTargetFreqConv2 := 0.0;
		rTargetFreqRot1 := 0.0;
		rTargetFreqRot2 := 0.0;

		// Сброс подстадий запуска и остановки
		nStartingSubstage := 0;
		nStoppingSubstage := 0;

		// Сброс таймеров запуска и остановки
		fbTimerStarting(IN := FALSE);
		fbTimerStopping(IN := FALSE);

		// Тормоза активны (удерживают механизм)
		Dumper.qxBreakerConveyor := FALSE;

		IF xStartCommand THEN
			STAGE := PRESTART_ALARM;
		END_IF;

	PRESTART_ALARM:
		// Проверка команды остановки во время предпусковой сигнализации
		IF xStopCommand THEN
			// Прервать предпусковую сигнализацию и вернуться в IDLE
			STAGE := E_StageWithPreStartAlarm.IDLE;
		ELSIF Dumper.fbPreStartAlarm.qxComplete THEN
			STAGE := E_StageWithPreStartAlarm.STARTING;
		END_IF;

	E_StageWithPreStartAlarm.STARTING:
		// Проверка команды остановки во время запуска
		IF xStopCommand THEN
			// Прервать запуск и перейти к процедуре остановки
			STAGE := E_StageWithPreStartAlarm.WORK;
			nStartingSubstage := 0;
			nStoppingSubstage := 1; // Начать процедуру остановки
			fbTimerStarting(IN := FALSE); // Сброс таймера
		END_IF;

		// Таймер ожидания полного запуска секции
		fbTimerStarting(
			IN := TRUE,
			PT := TIME_AFTER_START_DUMPER
		);

		// Последовательный запуск: Тормоза → Обратная связь → VFD → Разгон
		CASE nStartingSubstage OF
			0: // RELEASE_BRAKE - Отпускание тормозов
				// Включить сигнал тормоза (1 = тормоз отпущен)
				Dumper.qxBreakerConveyor := TRUE;
				Dumper.qxBreakerRotation := TRUE;

				// Переход к следующей подстадии
				nStartingSubstage := 1;

			1: // WAIT_BRAKE_FEEDBACK - Ожидание обратной связи тормозов
				// Получить обратную связь реле тормоза
				IF Dumper.fbBreakerConveyor.qxSignal THEN
					// Обратная связь получена, переходим к запуску VFD
					nStartingSubstage := 2;
				END_IF;

			2: // START_VFD - Запуск VFD (контакторы управляются отдельно через cmdBuildCircuitOn/Off)
				// Команда ПУСК на частотный преобразователь (TRUE = ПУСК)
				Dumper.MotorConveyor[1].VFD.qxStart := TRUE;
				Dumper.MotorConveyor[2].VFD.qxStart := TRUE;

				// Установка целевой частоты
				// (FB_FrequencyControl автоматически выберет плавный или прямой пуск через irStep)
				rTargetFreqConv1 := MOTOR_FREQUENCY_DUMPER_CONVEYOR;
				rTargetFreqConv2 := MOTOR_FREQUENCY_DUMPER_CONVEYOR;

				// Если оба VFD запущены (обратная связь), переходим к следующей подстадии
				IF Dumper.MotorConveyor[1].VFD.fbStateIsWorking.qxSignal
					AND Dumper.MotorConveyor[2].VFD.fbStateIsWorking.qxSignal
				THEN
					IF VFD_SMOOTH_SET_FREQUENCY THEN
						// Плавный пуск: переходим к разгону
						nStartingSubstage := 3;
					ELSE
						// Прямой пуск: сразу в режим WORK (частота уже установлена через большой шаг)
						STAGE := E_StageWithPreStartAlarm.WORK;
						nStartingSubstage := 0;
						fbTimerStarting(IN := FALSE); // Сброс таймера
					END_IF;
				END_IF;

			3: // RAMPING - Разгон частоты до рабочей
				// Команды запуска VFD остаются активными (TRUE = ПУСК)
				Dumper.MotorConveyor[1].VFD.qxStart := TRUE;
				Dumper.MotorConveyor[2].VFD.qxStart := TRUE;

				// Задание целевой частоты (передается в FB_FrequencyControl)
				rTargetFreqConv1 := MOTOR_FREQUENCY_DUMPER_CONVEYOR;
				rTargetFreqConv2 := MOTOR_FREQUENCY_DUMPER_CONVEYOR;

				// Переход в режим WORK при достижении целевой частоты
				// Используется регулирование частоты с синхронизацией
				IF Dumper.MotorConveyor[1].VFD.rActualFrequency >= MOTOR_FREQUENCY_DUMPER_CONVEYOR - VFD_FREQUENCY_INACCURANCY
					AND Dumper.MotorConveyor[2].VFD.rActualFrequency >= MOTOR_FREQUENCY_DUMPER_CONVEYOR - VFD_FREQUENCY_INACCURANCY
				THEN
					STAGE := E_StageWithPreStartAlarm.WORK;
					nStartingSubstage := 0; // Сброс для следующего запуска
					fbTimerStarting(IN := FALSE); // Сброс таймера
				END_IF;
		END_CASE;

	E_StageWithPreStartAlarm.WORK:
		// Нормальная работа или штатная остановка через подстадии
		CASE nStoppingSubstage OF
			0: // Нормальная работа
				// Сброс таймера остановки
				fbTimerStopping(IN := FALSE);

				// Обновление целевой частоты конвейера в ручном режиме
				IF Dumper.eStateRemote = E_StateRemote.Manual THEN
					rTargetFreqConv1 := MOTOR_FREQUENCY_DUMPER_CONVEYOR;
					rTargetFreqConv2 := MOTOR_FREQUENCY_DUMPER_CONVEYOR;
				END_IF;

				IF xStopCommand THEN
					// Начать штатную остановку
					nStoppingSubstage := 1;
				END_IF;

			1: // SET_FREQUENCY_ZERO - Установка частоты 0 на аналоговый выход
				// Запуск таймера остановки (тайм-аут на остановку секции)
				fbTimerStopping(
					IN := TRUE,
					PT := TIME_TIMEOUT_STOP_DUMPER
				);

				// Установить целевую частоту 0
				// (FB_FrequencyControl автоматически выберет плавную или прямую остановку через irStep)
				rTargetFreqConv1 := 0.0;
				rTargetFreqConv2 := 0.0;
				rTargetFreqRot1 := 0.0;
				rTargetFreqRot2 := 0.0;

				// Команды пуска VFD остаются активными (TRUE = ПУСК)
				// VFD продолжают работать, но частота снижается
				Dumper.MotorConveyor[1].VFD.qxStart := FALSE; // TODO ВРЕМЕННО
				Dumper.MotorConveyor[2].VFD.qxStart := FALSE;

				// Переход к следующей подстадии
				nStoppingSubstage := 2;

			2: // WAIT_FREQUENCY_ZERO - Ожидание подтверждения частоты 0 с аналогового входа
				// Ждём, пока фактическая частота (с аналогового входа) не снизится до 0 (+/- 2 Гц)
				IF Dumper.MotorConveyor[1].VFD.rActualFrequency <= 2.0
					AND Dumper.MotorConveyor[2].VFD.rActualFrequency <= 2.0
				THEN
					// Частота подтверждена на 0, переходим к остановке VFD
					nStoppingSubstage := 3;
				END_IF;

			3: // STOP_VFD - Остановка VFD (снятие команды пуска)
				// Отключить команду пуска на VFD (FALSE = СТОП)
				Dumper.MotorConveyor[1].VFD.qxStart := FALSE;
				Dumper.MotorConveyor[2].VFD.qxStart := FALSE;

				// Переход к ожиданию обратной связи VFD
				nStoppingSubstage := 4;

			4: // WAIT_VFD_STOP - Ожидание остановки VFD (обратная связь)
				// Проверить обратную связь VFD о выключении
				IF NOT Dumper.MotorConveyor[1].VFD.fbStateIsWorking.qxSignal
					AND NOT Dumper.MotorConveyor[2].VFD.fbStateIsWorking.qxSignal
				THEN
					// VFD выключены, переход к активации тормозов
					nStoppingSubstage := 5;
				END_IF;

			5: // ACTIVATE_BRAKE - Активация тормозов
				// Включение таймера на задержку тормоза
				tonTimerEnableBreakerConveyor(IN:= TRUE, PT:=T#5S);

				IF tonTimerEnableBreakerConveyor.Q THEN // Снять сигнал с тормоза после таймера (поставить на тормоз: FALSE = активен)
					Dumper.qxBreakerConveyor := FALSE;
					Dumper.qxBreakerRotation := FALSE;
					tonTimerEnableBreakerConveyor(IN:= FALSE);
					// Переход к завершению остановки
					nStoppingSubstage := 6;
				END_IF;
			6: // WAIT_BRAKE_FEEDBACK - Переход в IDLE
				// Сброс таймера остановки (успешная остановка)
				fbTimerStopping(IN := FALSE);

				STAGE := E_StageWithPreStartAlarm.IDLE;
				nStoppingSubstage := 0;
		END_CASE;

	E_StageWithPreStartAlarm.ERROR:
		// Состояние ошибки - аварийная остановка и ожидание сброса
		// (используется при серьезных неисправностях, не для штатной остановки)

		// Аварийная остановка: команда СТОП на VFD (FALSE = СТОП)
		Dumper.MotorConveyor[1].VFD.qxStart := FALSE;
		Dumper.MotorConveyor[2].VFD.qxStart := FALSE;
		Dumper.MotorRotation[1].VFD.qxStart := FALSE;
		Dumper.MotorRotation[2].VFD.qxStart := FALSE;
		Dumper.MotorRotation[1].qxVFDReverseStart := FALSE;
		Dumper.MotorRotation[2].qxVFDReverseStart := FALSE;

		// Сброс целевых частот
		rTargetFreqConv1 := 0.0;
		rTargetFreqConv2 := 0.0;
		rTargetFreqRot1 := 0.0;
		rTargetFreqRot2 := 0.0;

		// Активировать тормоза
		Dumper.qxBreakerConveyor := FALSE;
		Dumper.qxBreakerRotation := FALSE;

		// Разборка схем контакторов (аварийная остановка)
		IF Dumper.eStateRemote = E_StateRemote.Auto THEN
			xCircuitBuilt := FALSE;
			xCircuitBuiltRotation := FALSE;
		END_IF;
		// Сброс подстадий для следующего запуска
		nStartingSubstage := 0;
		nStoppingSubstage := 0;
		nRotationSubstage := 0;

		// Сброс таймеров
		fbTimerStarting(IN := FALSE);
		fbTimerStopping(IN := FALSE);
		fbTimerRotation(IN := FALSE);
		tonTimerEnableBreakerConveyor(IN := FALSE);
		tonTimerEnableBreakerRotation(IN:= FALSE);
		// Контакторы управляются отдельно через импульсные команды
		// cmdBuildCircuitOn/Off (см. секцию УПРАВЛЕНИЕ КОНТАКТОРАМИ)

		// Сброс ошибки и переход в IDLE при отсутствии ошибок
		// Для выхода из ERROR требуется:
		// 1. Команда сброса (xReset)
		// 2. Снятие сигнала аварийной остановки (NOT xEmergencyStop)
		// 3. Кнопка аварийной остановки отпущена (NC контакт: TRUE = кнопка отпущена)
		// 4. Отсутствие ошибок оборудования (NOT Dumper.xStateFailure)
		IF xReset AND NOT xEmergencyStop AND Dumper.fbBtnEmergencyStop.qxSignal AND NOT Dumper.xStateFailure THEN
			STAGE := E_StageWithPreStartAlarm.IDLE;
		END_IF
END_CASE;

// ========================================
// ПРОВЕРКА СИНХРОНИЗАЦИИ МОТОРОВ КОНВЕЙЕРА
// ========================================

// Проверка что оба ЧРП конвейера готовы и запущены (обратная связь)
xVFDsReady := Dumper.MotorConveyor[1].VFD.fbStateIsWorking.qxSignal
           AND Dumper.MotorConveyor[2].VFD.fbStateIsWorking.qxSignal;

// Проверка синхронизации текущих частот (разница не превышает допуск)
xFrequenciesSynchronized := ABS(Dumper.MotorConveyor[1].VFD.Frequency.qrCurrentFrequency
                              - Dumper.MotorConveyor[2].VFD.Frequency.qrCurrentFrequency)
                              <= VFD_FREQUENCY_SYNC_TOLERANCE;

// Общее условие для продолжения плавного разгона
// Разгон продолжается только если оба ЧРП запущены И частоты синхронизированы
xConditionToProceed := xVFDsReady AND xFrequenciesSynchronized;

// ========================================
// ОБРАБОТКА ЧАСТОТЫ (после установки целевых значений в CASE)
// ========================================

// Моторы конвейера
Dumper.MotorConveyor[1].VFD.Frequency(
	irMaxFrequency := VFD_FREQUENCY_MAX,
	// Если плавный пуск - используем шаг, иначе - большой шаг для мгновенной установки
	irStep := SEL(VFD_SMOOTH_SET_FREQUENCY, VFD_FREQ_MAX_RANGE, VFD_FREQUENCY_STEP),
	rTargetFrequency := rTargetFreqConv1,
	xPulse := PULSE_RTRIG.Q,
	xConditionToProceed := xConditionToProceed // Синхронизация с мотором 2
);
// qrCurrentFrequency передается напрямую в fbAnalogOutput.rEngValue

Dumper.MotorConveyor[2].VFD.Frequency(
	irMaxFrequency := VFD_FREQUENCY_MAX,
	// Если плавный пуск - используем шаг, иначе - большой шаг для мгновенной установки
	irStep := SEL(VFD_SMOOTH_SET_FREQUENCY, VFD_FREQ_MAX_RANGE, VFD_FREQUENCY_STEP),
	rTargetFrequency := rTargetFreqConv2,
	xPulse := PULSE_RTRIG.Q,
	xConditionToProceed := xConditionToProceed // Синхронизация с мотором 1
);
// qrCurrentFrequency передается напрямую в fbAnalogOutput.rEngValue

// Моторы поворота
Dumper.MotorRotation[1].VFD.Frequency(
	irMaxFrequency := VFD_FREQUENCY_MAX,
	// Если плавный пуск - используем шаг, иначе - большой шаг для мгновенной установки
	irStep := SEL(VFD_SMOOTH_SET_FREQUENCY, VFD_FREQ_MAX_RANGE, VFD_FREQUENCY_STEP),
	rTargetFrequency := rTargetFreqRot1,
	xPulse := PULSE_RTRIG.Q,
	xConditionToProceed := TRUE
);
// qrCurrentFrequency передается напрямую в fbAnalogOutput.rEngValue

Dumper.MotorRotation[2].VFD.Frequency(
	irMaxFrequency := VFD_FREQUENCY_MAX,
	// Если плавный пуск - используем шаг, иначе - большой шаг для мгновенной установки
	irStep := SEL(VFD_SMOOTH_SET_FREQUENCY, VFD_FREQ_MAX_RANGE, VFD_FREQUENCY_STEP),
	rTargetFrequency := rTargetFreqRot2,
	xPulse := PULSE_RTRIG.Q,
	xConditionToProceed := TRUE
);
// qrCurrentFrequency передается напрямую в fbAnalogOutput.rEngValue

// Вывод текущей стадии
eStage := STAGE;

// ========================================
// УПРАВЛЕНИЕ КОНТАКТОРАМИ
// ========================================

// РУЧНОЙ РЕЖИМ (Manual):
// - Схема управляется ТОЛЬКО импульсными командами cmdBuildCircuitOn/Off
// - Автоматическая сборка/разборка схемы ОТКЛЮЧЕНА
//
// АВТОМАТИЧЕСКИЙ РЕЖИМ (Auto/Remote):
// - Схема собирается АВТОМАТИЧЕСКИ при отсутствии ошибок секции:
//   * Нет ошибок по датчикам безопасности (FC_Dumper_GetErrorSensors = FALSE)
//   * Секция НЕ в стадии ERROR
// - Схема разбирается АВТОМАТИЧЕСКИ при появлении ошибок или переходе в ERROR

IF Dumper.eStateRemote = E_StateRemote.Manual THEN
	// РУЧНОЙ РЕЖИМ - Обработка импульсных команд сборки/разборки схемы конвейера
	// cmdBuildCircuitOn - собрать схему (включить контакторы)
	// cmdBuildCircuitOff - разобрать схему (выключить контакторы)
	IF Dumper.cmdBuildCircuitOn THEN
		xCircuitBuilt := TRUE;
		Dumper.cmdBuildCircuitOn := FALSE; // Сброс импульсной команды
	ELSIF Dumper.cmdBuildCircuitOff THEN
		xCircuitBuilt := FALSE;
		Dumper.cmdBuildCircuitOff := FALSE; // Сброс импульсной команды
	END_IF;
ELSIF Dumper.eStateRemote = E_StateRemote.Auto THEN
	// АВТОМАТИЧЕСКИЙ РЕЖИМ - Автоматическая сборка схемы при отсутствии ошибок
	// Собираем схему если:
	// 1. Нет ошибок по датчикам безопасности
	// 2. Секция НЕ в стадии ERROR
	IF NOT FC_Dumper_GetErrorSensors(Dumper := Dumper) AND STAGE <> E_StageWithPreStartAlarm.ERROR THEN
		xCircuitBuilt := TRUE;
	ELSE
		xCircuitBuilt := FALSE;
	END_IF;
END_IF;

// Моторы конвейера - управление контакторами через состояние схемы
Dumper.MotorConveyor[1].qxKM_Power := xCircuitBuilt;
Dumper.MotorConveyor[2].qxKM_Power := xCircuitBuilt;

IF Dumper.eStateRemote = E_StateRemote.Manual THEN
	// РУЧНОЙ РЕЖИМ - Обработка импульсных команд сборки/разборки схемы поворота
	// cmdBuildCircuitOnRotation - собрать схему поворота (включить контакторы)
	// cmdBuildCircuitOffRotation - разобрать схему поворота (выключить контакторы)
	IF Dumper.cmdBuildCircuitOnRotation THEN
		xCircuitBuiltRotation := TRUE;
		Dumper.cmdBuildCircuitOnRotation := FALSE; // Сброс импульсной команды
	ELSIF Dumper.cmdBuildCircuitOffRotation THEN
		xCircuitBuiltRotation := FALSE;
		Dumper.cmdBuildCircuitOffRotation := FALSE; // Сброс импульсной команды
	END_IF;
ELSIF Dumper.eStateRemote = E_StateRemote.Auto THEN
	// АВТОМАТИЧЕСКИЙ РЕЖИМ - Автоматическая сборка схемы поворота при отсутствии ошибок
	// Собираем схему если:
	// 1. Нет ошибок по датчикам безопасности
	// 2. Секция НЕ в стадии ERROR
	IF NOT FC_Dumper_GetErrorSensors(Dumper := Dumper) AND STAGE <> E_StageWithPreStartAlarm.ERROR THEN
		xCircuitBuiltRotation := TRUE;
	ELSE
		xCircuitBuiltRotation := FALSE;
	END_IF;
END_IF;

// Моторы поворота - управление контакторами через состояние схемы
Dumper.MotorRotation[1].qxKM_Power := xCircuitBuiltRotation;
Dumper.MotorRotation[2].qxKM_Power := xCircuitBuiltRotation;

// ========================================
// УПРАВЛЕНИЕ МОТОРАМИ ПОВОРОТА
// ========================================

// Обработка команд поворота в зависимости от режима управления

IF xLocalMode THEN
	// ========== МЕСТНЫЙ РЕЖИМ (ПМУ) ==========
	// В местном режиме: поворот работает ПОКА ЗАЖАТА КНОПКА

	// ПУСК поворота влево - при зажатой кнопке и отсутствии активного поворота
	IF Dumper.fbBtnTurnLeft.qxSignal AND nRotationSubstage = 0 THEN
		// Можем начать поворот влево только если:
		// 1. Левый концевик НЕ сработал (qxSignal = TRUE означает концевик в норме, не нажат)
		// 2. Нет активного поворота
		IF Dumper.fbEndSwitchLeft.qxSignal THEN
			xRotationLeftActive := TRUE;
			xRotationRightActive := FALSE;
			nRotationSubstage := 1; // Начать последовательность запуска
		END_IF;
		// Если концевик сработал (qxSignal = FALSE), команда игнорируется
	END_IF;

	// ПУСК поворота вправо - при зажатой кнопке и отсутствии активного поворота
	IF Dumper.fbBtnTurnRight.qxSignal AND nRotationSubstage = 0 THEN
		// Можем начать поворот вправо только если:
		// 1. Правый концевик НЕ сработал (qxSignal = TRUE означает концевик в норме, не нажат)
		// 2. Нет активного поворота
		IF Dumper.fbEndSwitchRight.qxSignal THEN
			xRotationRightActive := TRUE;
			xRotationLeftActive := FALSE;
			nRotationSubstage := 1; // Начать последовательность запуска
		END_IF;
		// Если концевик сработал (qxSignal = FALSE), команда игнорируется
	END_IF;

	// ОСТАНОВКА поворота - когда кнопка отпущена или достигнут концевик
	IF nRotationSubstage >= 1 AND nRotationSubstage <= 4 THEN
		// Условия остановки:
		// 1. Кнопка отпущена (для левого поворота - кнопка влево отпущена, для правого - кнопка вправо)
		// 2. Достигнут концевик
		IF (xRotationLeftActive AND (NOT Dumper.fbBtnTurnLeft.qxSignal OR NOT Dumper.fbEndSwitchLeft.qxSignal))
			OR (xRotationRightActive AND (NOT Dumper.fbBtnTurnRight.qxSignal OR NOT Dumper.fbEndSwitchRight.qxSignal))
		THEN
			// Начать последовательность остановки
			nRotationSubstage := 5;
		END_IF;
	END_IF;

ELSE
	// ========== ДИСТАНЦИОННЫЙ РЕЖИМ (SCADA) ==========
	// В дистанционном режиме: импульсные команды от АСУТП

	// Обработка команды поворота влево
	IF Dumper.cmdTurnLeft AND nRotationSubstage = 0 THEN
		// Можем начать поворот влево только если:
		// 1. Левый концевик НЕ сработал (qxSignal = TRUE означает концевик в норме, не нажат)
		// 2. Нет активного поворота
		IF Dumper.fbEndSwitchLeft.qxSignal THEN
			xRotationLeftActive := TRUE;
			xRotationRightActive := FALSE;
			nRotationSubstage := 1; // Начать последовательность запуска
		END_IF;
		// Если концевик сработал (qxSignal = FALSE), команда игнорируется
	END_IF;

	// Обработка команды поворота вправо
	IF Dumper.cmdTurnRight AND nRotationSubstage = 0 THEN
		// Можем начать поворот вправо только если:
		// 1. Правый концевик НЕ сработал (qxSignal = TRUE означает концевик в норме, не нажат)
		// 2. Нет активного поворота
		IF Dumper.fbEndSwitchRight.qxSignal THEN
			xRotationRightActive := TRUE;
			xRotationLeftActive := FALSE;
			nRotationSubstage := 1; // Начать последовательность запуска
		END_IF;
		// Если концевик сработал (qxSignal = FALSE), команда игнорируется
	END_IF;

	// Условия остановки поворота:
	// 1. Достигнут концевик
	// 2. Импульсная команда остановки (cmdStopRotation)
	IF nRotationSubstage >= 1 AND nRotationSubstage <= 4 THEN
		// Проверка условий остановки
		IF (xRotationLeftActive AND NOT Dumper.fbEndSwitchLeft.qxSignal)
			OR (xRotationRightActive AND NOT Dumper.fbEndSwitchRight.qxSignal)
			OR Dumper.cmdStopRotation
		THEN
			// Начать последовательность остановки
			nRotationSubstage := 5;
		END_IF;
	END_IF;

	// Сброс импульсных команд от АСУТП
	IF Dumper.cmdTurnLeft THEN
		Dumper.cmdTurnLeft := FALSE;
	END_IF;
	IF Dumper.cmdTurnRight THEN
		Dumper.cmdTurnRight := FALSE;
	END_IF;
	IF Dumper.cmdStopRotation THEN
		Dumper.cmdStopRotation := FALSE;
	END_IF;
END_IF;

// Автомат управления поворотом с подстадиями
CASE nRotationSubstage OF
	0: // IDLE - Нет активного поворота
		// Сброс таймера поворота
		fbTimerRotation(IN := FALSE);
		tonTimerEnableBreakerRotation.IN :=  FALSE;
		// Остановка VFD
		Dumper.MotorRotation[1].VFD.qxStart := FALSE;
		Dumper.MotorRotation[2].VFD.qxStart := FALSE;
		Dumper.MotorRotation[1].qxVFDReverseStart := FALSE;
		Dumper.MotorRotation[2].qxVFDReverseStart := FALSE;

		// Активация тормоза поворота
		Dumper.qxBreakerRotation := FALSE;

		// Сброс целевой частоты
		rTargetFreqRot1 := 0.0;
		rTargetFreqRot2 := 0.0;

		// Сброс флагов поворота
		xRotationLeftActive := FALSE;
		xRotationRightActive := FALSE;

	1: // RELEASE_BRAKE - Отпускание тормоза поворота
		// Запуск таймера поворота (тайм-аут на выполнение команды поворота)
		fbTimerRotation(
			IN := TRUE,
			PT := TIME_TIMEOUT_ROTATION_DUMPER
		);

		// Отпустить тормоз (1 = тормоз отпущен)
		Dumper.qxBreakerRotation := TRUE;

		// Переход к следующей подстадии
		nRotationSubstage := 2;

	2: // WAIT_BRAKE_FEEDBACK - Ожидание обратной связи тормоза
		// Ждём обратную связь реле тормоза
		IF Dumper.fbBreakerRotation.qxSignal THEN
			// Обратная связь получена, переходим к запуску VFD
			nRotationSubstage := 3;
		END_IF;

	3: // START_VFD - Запуск VFD поворота
		IF xRotationLeftActive THEN
			// Поворот влево - запуск в прямом направлении
			Dumper.MotorRotation[1].qxVFDReverseStart := FALSE;
			Dumper.MotorRotation[2].qxVFDReverseStart := FALSE;
			Dumper.MotorRotation[1].VFD.qxStart := TRUE;
			Dumper.MotorRotation[2].VFD.qxStart := TRUE;

		ELSIF xRotationRightActive THEN
			// Поворот вправо - запуск в режиме реверса
			Dumper.MotorRotation[1].VFD.qxStart := FALSE;
			Dumper.MotorRotation[2].VFD.qxStart := FALSE;
			Dumper.MotorRotation[1].qxVFDReverseStart := TRUE;
			Dumper.MotorRotation[2].qxVFDReverseStart := TRUE;
		END_IF;

		// Установка целевой частоты
		rTargetFreqRot1 := MOTOR_FREQUENCY_DUMPER_ROTATION;
		rTargetFreqRot2 := MOTOR_FREQUENCY_DUMPER_ROTATION;

		// Проверка запуска VFD (обратная связь)
		IF Dumper.MotorRotation[1].VFD.fbStateIsWorking.qxSignal
			AND Dumper.MotorRotation[2].VFD.fbStateIsWorking.qxSignal
		THEN
			// VFD запущены, переходим в режим работы
			nRotationSubstage := 4;
		END_IF;

	4: // WORKING - Моторы поворота работают
		// Поддержка целевой частоты
		rTargetFreqRot1 := MOTOR_FREQUENCY_DUMPER_ROTATION;
		rTargetFreqRot2 := MOTOR_FREQUENCY_DUMPER_ROTATION;

	5: // SET_FREQUENCY_ZERO - Установка частоты 0 на аналоговый выход
		// Установить целевую частоту 0
		// (FB_FrequencyControl автоматически выберет плавную или прямую остановку через irStep)
		rTargetFreqRot1 := 0.0;
		rTargetFreqRot2 := 0.0;

		// Команды пуска VFD остаются активными (VFD продолжают работать, но частота снижается)
		// Переход к следующей подстадии
		nRotationSubstage := 6;

	6: // WAIT_FREQUENCY_ZERO - Ожидание подтверждения частоты 0 с аналогового входа
		// Ждём, пока фактическая частота (с аналогового входа) не снизится до 0 (+/- 2 Гц)
//		IF Dumper.MotorRotation[1].VFD.rActualFrequency <= 2.0
//			AND Dumper.MotorRotation[2].VFD.rActualFrequency <= 2.0
//		THEN
			// Частота подтверждена на 0, переходим к остановке VFD
			nRotationSubstage := 7;
//		END_IF;

	7: // STOP_VFD - Остановка VFD поворота (снятие команды пуска)
		// Отключить команду пуска на VFD (FALSE = СТОП)
		Dumper.MotorRotation[1].VFD.qxStart := FALSE;
		Dumper.MotorRotation[2].VFD.qxStart := FALSE;
		Dumper.MotorRotation[1].qxVFDReverseStart := FALSE;
		Dumper.MotorRotation[2].qxVFDReverseStart := FALSE;

		// Переход к ожиданию обратной связи VFD
		nRotationSubstage := 8;

	8: // WAIT_VFD_STOP - Ожидание остановки VFD (обратная связь)
		// Проверить обратную связь VFD о выключении
		IF NOT Dumper.MotorRotation[1].VFD.fbStateIsWorking.qxSignal
			AND NOT Dumper.MotorRotation[2].VFD.fbStateIsWorking.qxSignal
		THEN
			// VFD выключены, переход к активации тормоза
			nRotationSubstage := 9;
		END_IF;

	9: // ACTIVATE_BRAKE - Активация тормоза
		tonTimerEnableBreakerRotation(IN:= TRUE, PT:=T#3S);
		IF tonTimerEnableBreakerRotation.Q THEN
			// Снять сигнал с тормоза (поставить на тормоз: FALSE = активен)
			Dumper.qxBreakerRotation := FALSE;
        	tonTimerEnableBreakerRotation(IN:= FALSE);
			// Сброс таймера поворота (успешное выполнение команды)
			fbTimerRotation(IN := FALSE);
			// Переход в IDLE
			nRotationSubstage := 0;
		END_IF;
END_CASE;

// ========================================
// ОБНОВЛЕНИЕ РЕЖИМА УПРАВЛЕНИЯ
// ========================================

// Если установлен местный режим (xLocalMode = TRUE), то переводим в Manual
// Manual может работать как дистанционно (от SCADA), так и местно (от ПМУ)
IF xLocalMode THEN
	Dumper.eStateRemote := E_StateRemote.Manual;
END_IF;

// ========================================
// ПЕРЕДАЧА СОСТОЯНИЙ ДЛЯ SCADA
// ========================================

// Приоритет проверки: от более критичных к менее критичным
IF STAGE = E_StageWithPreStartAlarm.ERROR THEN
	// Ошибка без активной работы
	eStageToSCADA := E_ScadaStatesDevice.ERROR;

ELSIF STAGE = E_StageWithPreStartAlarm.WORK AND Dumper.xStateFailure THEN
	// TODO: Секция работает с аварией (требует уточнения логики)
	// Обычно при ошибке должна быть остановка, но оставляем для будущей реализации
	eStageToSCADA := E_ScadaStatesDevice.WORK_WITH_ERROR;

ELSIF STAGE = E_StageWithPreStartAlarm.WORK AND Dumper.xStateWarning THEN
	// Секция работает с предупреждением
	eStageToSCADA := E_ScadaStatesDevice.WORK_WITH_WARNING;

ELSIF STAGE = E_StageWithPreStartAlarm.WORK THEN
	// Секция работает в норме (нет ошибок и предупреждений)
	eStageToSCADA := E_ScadaStatesDevice.WORK;

ELSIF Dumper.xStateStarting THEN
	// Секция в процессе запуска (предпусковая сигнализация или разгон)
	eStageToSCADA := E_ScadaStatesDevice.STARTING;

ELSIF STAGE = E_StageWithPreStartAlarm.IDLE AND Dumper.xStateWarning THEN
	// Предупреждение без активной работы
	eStageToSCADA := E_ScadaStatesDevice.WARNING;

ELSIF STAGE = E_StageWithPreStartAlarm.IDLE AND Dumper.xStateFailure THEN
	// Секция неготова к запуску (есть ошибки)
	eStageToSCADA := E_ScadaStatesDevice.NOT_READY;

ELSE
	// Секция готова к запуску (IDLE, нет ошибок и предупреждений)
	eStageToSCADA := E_ScadaStatesDevice.READY;

END_IF;

// Передача состояний режима управления
Dumper.xStateRemoteAuto := Dumper.eStateRemote = E_StateRemote.Auto;
Dumper.xStateRemoteManual := Dumper.eStateRemote = E_StateRemote.Manual;
Dumper.xStateRemoteRepair := Dumper.eStateRemote = E_StateRemote.Repair;

END_FUNCTION_BLOCK

(* ---- FB_FrequencySimulation.st ---- *)
FUNCTION_BLOCK FB_FrequencySimulation
VAR_INPUT
    xProceed : BOOL;        // Флаг работы ФБ (TRUE = работает, FALSE = остановлен)
    irTarget : REAL;        // Цель частоты
    irStep : REAL;          // Шаг изменения за цикл
END_VAR
VAR_OUTPUT
    irInputModule : REAL;   // Текущие показания (симуляция обратной связи)
END_VAR
VAR
    rDifference : REAL;     // Разница между целью и текущим значением
END_VAR
// Проверяем флаг работы
IF xProceed THEN
    // Вычисляем разницу между целевым и текущим значением
    rDifference := irTarget - irInputModule;

    // Проверяем, не достигли ли мы уже цели
    IF ABS(rDifference) <= ABS(irStep) THEN
        // Если разница меньше или равна шагу, устанавливаем точное значение
        irInputModule := irTarget;
    ELSE
        // Иначе двигаемся к цели с заданным шагом
        IF rDifference > 0 THEN
            // Цель выше текущего значения - увеличиваем
            irInputModule := irInputModule + ABS(irStep);
        ELSE
            // Цель ниже текущего значения - уменьшаем
            irInputModule := irInputModule - ABS(irStep);
        END_IF;
    END_IF;
ELSE
    // Если ЧРП не работает, сбрасываем частоту в 0
    irInputModule := 0.0;
END_IF;

END_FUNCTION_BLOCK
